FUNCTION F_GetTransportTubeStatuses : ST_TransportTubeStatuses
VAR_INPUT
	eTransportTube : T_TransportTube;
END_VAR
VAR
	fbTT : REFERENCE TO FB_TransportTube;
	stStatus : ST_TransportTubeStatuses := ();
END_VAR

fbTT REF= F_GetTransportTube(eTransportTube);

stStatus.bIonPumpOn := fbTT.q_stConfig.stDevices.refIonPump.q_xHVEna_DO;
stStatus.bGateValveOpen := fbTT.q_stConfig.stDevices.refGateValve.M_IsOpen();
stStatus.fPiraniVal := fbTT.q_stConfig.stDevices.refPiraniGauge.PG.rPRESS;
stStatus.fColdCathodeVal := fbTT.q_stConfig.stDevices.refColdCathode.IG.rPRESS;

F_GetTransportTubeStatuses := stStatus;

END_FUNCTION

(* stored: Version 1.1.0.1, ProductVersion 3.1.4022.17
   POU F_GetTransportTubeStatuses: Id {09b6220d-41cc-0b3f-3e37-f70d9621ad78}, SpecialFunc None *)
